// TwinCAT 3 PLC project PLC
// ProgramVersion: 3.1.4026.22
// libraries:
//   Tc2_MC2, * (Beckhoff Automation GmbH)
//   Tc2_Standard, * (Beckhoff Automation GmbH)
//   Tc2_System, * (Beckhoff Automation GmbH)
//   Tc2_Utilities, * (Beckhoff Automation GmbH)
// project tree:
//   DUTs/ E_AxisState.TcDUT (not stored)
//   / PlcTask.TcTTO
//   POUs/FBs/ FB_SimpleAxis.TcPOU (not stored)
//   POUs/ MAIN.TcPOU (not stored), P_ReverseSequence.TcPOU (not stored), P_ScannerSim.TcPOU (not stored), P_ScopeServer.TcPOU
// real-time tasks:
//   TASK PlcTask: cycle T#10ms, priority 20, ADS port 350
// motion (NC):
//   TASK NC-Task 1 SAF: cycle T#2ms, priority 4, ADS port 501
//   TASK NC-Task 1 SVB: cycle T#10ms, priority 8, ADS port 511
//   AXIS Axis 1 (id 1)
//     OtherSettings: AllowMotionCmdToSlave=true
//     encoder EncType=1
//     drive DrvType=5
//       Analog: TorqueSetpointScale=10, ScaleFactorActTorque=0.1
//       TimeComp: TaskDelayCycles=1
//     controller CtrType=1
//       CtrPara: PriorControlFactor=1
//         Observer: BandWidth=20
// variable links:
//   PLC/PLC Instance <-> NC-Task 1 SAF/Axes/Axis 1
//     PlcTask Inputs/P_ReverseSequence.fbAxis.stAxis.NcToPlc <-> Outputs/ToPlc
//     PlcTask Outputs/P_ReverseSequence.fbAxis.stAxis.PlcToNc <-> Inputs/FromPlc

CONFIGURATION PLC
    RESOURCE PLC ON TwinCAT3
        TASK PlcTask(INTERVAL := T#10ms, PRIORITY := 20);
        PROGRAM MAIN WITH PlcTask : MAIN;
    END_RESOURCE
END_CONFIGURATION

// ---- POUs/P_ScopeServer.TcPOU
PROGRAM P_ScopeServer
VAR

END_VAR

END_PROGRAM
